PROGRAM PRG_TEST
VAR
	HeatingCurve_Test : FC_HeatingCurve_Test;
	FanControlTest : FB_FanControl_Test;
END_VAR

TcUnit.RUN();

END_PROGRAM

(* stored: Version 1.1.0.1, ProductVersion 3.1.4024.6
   POU PRG_TEST: Id {b7aacc06-295a-4dea-ac85-460d15a60691}, SpecialFunc None *)
